Omron Sysmac Studio project python_plc (Sysmac Studio 1.30.0.17, StandardProject)

# Controller new_Controller_0: NX1P2-1140DT1 version 1.13
Axis Sag_kol, settings changed from default: 
Axis Sol_kol, settings changed from default: AxisNumber=1, AxisType=ServoType, UnitsConversion=EnumElement5, UnitsNumerator=8388608, UnitsDenominator=360, MaxVelocity=18000, MaxJogVelocity=18000, MaxPositiveTorqueLimit=350.0, MaxNegativeTorqueLimit=350.0, CountMode=EnumElement2, ModuloMAXPosition=361, ModuloMINPosition=-1, EncoderTypes=Abs
Task PrimaryTask (priority 4, period or condition 2000): Program2
Library MTCP_NJ 1.3. (contents left out)

TYPE Modbus_Data : UNION
    Datas : ARRAY[0..1023] OF word;
    Datas_Dword : ARRAY[0..511] OF DWORD;  (* 4byte *)
    Datas_Lword : ARRAY[0..255] OF lword;  (* 8 byte *)
END_UNION END_TYPE
TYPE Servo : STRUCT
    mc_pwr_ready : BOOL;
    mc_pwr_busy : BOOL;
    mc_pwr_err : BOOL;
    mc_pwr_id : WORD;
    jog_positive_enable : BOOL;
    jog_negative_enable : BOOL;
    velocity : LREAL;
    acc_val : LREAL;
    dec_val : LREAL;
    jog_busy : BOOL;
    jog_aborted : BOOL;
    jog_error : BOOL;
    jog_error_id : WORD;
    position_enable : BOOL;
    position_val : LREAL;
    position_direction : _eMC_DIRECTION;
    position_done : BOOL;
    position_busy : BOOL;
    position_active : BOOL;
    position_aborted : BOOL;
    position_err : BOOL;
    position_err_id : word;
    reset_execute : BOOL;
    reset_busy : BOOL;
    reset_failure : BOOL;
    reset_err : BOOL;
    reset_err_id : WORD;
END_STRUCT END_TYPE
TYPE Srv : STRUCT
    Axis : _sAXIS_REF;
    pwr_enable : BOOL;
    pwr_busy : BOOL;
    pwr_err : BOOL;
    pwr_errid : WORD;
    pwr_status : BOOL;
    rst_enable : BOOL;
    rst_busy : BOOL;
    rst_failure : BOOL;
    rst_err : BOOL;
    rst_errid : WORD;
    rst_done : BOOL;
    parameter : _sAXIS_PARAM;
    read_enable : BOOL;
    read_busy : BOOL;
    read_aborted : BOOL;
    read_err : BOOL;
    read_errid : WORD;
    read_done : BOOL;
    move_enable : BOOL;
    move_position : LREAL;
    move_velocity : LREAL;
    move_acc : LREAL;
    move_dcc : LREAL;
    move_jerk : LREAL;
    move_direction : _eMC_DIRECTION;
    move_buffermode : _eMC_BUFFER_MODE;
    move_mode : _eMC_MOVE_MODE;
    move_busy : BOOL;
    move_active : BOOL;
    move_aborted : BOOL;
    move_err : BOOL;
    move_errid : WORD;
    move_done : BOOL;
    jog_pos_enable : BOOL;
    jog_neg_enable : BOOL;
    jog_velocity : LREAL;
    jog_acc : LREAL;
    jog_dcc : LREAL;
    jog_busy : bool;
    jog_aborted : bool;
    jog_err : bool;
    jog_errid : WORD;
    jog_errid_Copy : WORD;
    move_velocity_enable : BOOL;
    move_velocity_position : LREAL;
    move_velocity_velocity : LREAL;
    move_velocity_acc : LREAL;
    move_velocity_dcc : LREAL;
    move_velocity_jerk : LREAL;
    move_velocity_direction : _eMC_DIRECTION;
    move_velocity_buffermode : _eMC_BUFFER_MODE;
    move_velocity_continous : bool;
    move_velocity_busy : BOOL;
    move_velocity_active : BOOL;
    move_velocity_aborted : BOOL;
    move_velocity_err : BOOL;
    move_velocity_errid : WORD;
    move_velocity_done : BOOL;
    servo_start : BOOL;
    sync_move_start : bool;
    sync_move_buffer : _eMC_BUFFER_MODE;
    sync_move_inPosition : bool;
    sync_move_busy : bool;
    sync_move_active : bool;
    sync_move_aborted : bool;
    sync_move_error : bool;
    sync_move_errorid : WORD;
    sync_move_relative_start : bool;
    sync_move_relative_buffer : _eMC_BUFFER_MODE;
    sync_move_relative_invelocity : bool;
    sync_move_relative_active : bool;
    sync_move_relative_busy : bool;
    sync_move_relative_aborted : bool;
    sync_move_relative_error : bool;
    sync_move_relative_errorid : WORD;
    sync_move_relative_mode : _eMC_CMDPOS_MODE;
END_STRUCT END_TYPE
TYPE UDP_Data : UNION
    bytes : ARRAY[0..1999] OF BYTE;
    words : ARRAY[0..999] OF WORD;
    dwords : ARRAY[0..499] OF DWORD;
    lwords : ARRAY[0..249] OF LWORD;
END_UNION END_TYPE

VAR_GLOBAL CONSTANT
    Sol_kol : _sAXIS_REF;  (* at MC://_MC_AX[1] *)
END_VAR
VAR_GLOBAL
    register_array : Modbus_Data;
    Sistem_start : BOOL;  (* at BuiltInIO://cpu/#0/Input_Bit_00 *)
    Sistem_stop : BOOL;  (* at BuiltInIO://cpu/#0/Input_Bit_01 *)
    Reset : BOOL;  (* at BuiltInIO://cpu/#0/Input_Bit_02 *)
    Acil_Stop : BOOL;  (* at BuiltInIO://cpu/#0/Input_Bit_03 *)
END_VAR
VAR_GLOBAL CONSTANT
    Sag_kol : _sAXIS_REF;  (* at MC://_MC_AX[0] *)
END_VAR
VAR_GLOBAL
    statusword_s1 : WORD;  (* at ECAT://node#1/Statusword *)
    error_code_s1 : WORD;  (* at ECAT://node#1/Error code *)
    pos_act_s1 : DINT;  (* at ECAT://node#1/Position actual value *)
    trq_act_s1 : INT;  (* at ECAT://node#1/Torque actual value *)
    mode_s1 : SINT;  (* at ECAT://node#1/Modes of operation display *)
    digital_inputs_s1 : DWORD;  (* at ECAT://node#1/Digital inputs *)
END_VAR

PROGRAM Program0
VAR
    start : BOOL;
    sistem_calisiyor : BOOL;
    stop : BOOL;
    reset : BOOL;
    tcp_port_no : UINT := 0;
    tcp_port_add : STRING[15] := '192.168.0.100';
    dst_port : UINT := 6000;
    Trigger : BOOL;
    MTCP_Server_fc : MTCP_Server;
    Register_Modbus : ARRAY[0..1023] OF LREAL;
    coils : ARRAY[0..1023] OF BOOL;
    baglan2 : BOOL;
    MTCP_Client_Fn06_fb : MTCP_Client_Fn06;
    say : INT;
    ARADEGER : WORD;
    ARA2 : INT;
    fccnt : CTU;
    Servo_1_Hazir : BOOL;
    Servo_2_Hazir : bool;
    servo1_pwr : MC_Power;
    servo1_jog_fc : MC_MoveJog;
    servo1_move_abs_fc : MC_MoveAbsolute;
    servo2_pwr : MC_Power;
    servo2_move_abs_fc : MC_MoveAbsolute;
    servo1_reset_fc : MC_Reset;
    servo2_reset_fc : MC_Reset;
    baglan : bool;
    Register_Modbus_real : ARRAY[0..1023] OF real;
    ara : LINT;
    servo2_jog_fc : MC_MoveJog;
    run : BOOL;
    i : INT;
    tmp : LREAL;
    whatcdog : WORD := 9999;
    TCP_error : BOOL;
    TCP_ID : WORD;
    TCP_status : _eCONNECTION_STATE;
    tmp2 : LWORD;
    Status_notconnected : _eCONNECTION_STATE := _ESTABLISHED;
    fc_ton : TON;
    fc_ton1 : TON;
    fc_set : RS;
    fc_sr : SR;
    c : BOOL;
    testttt : REAL;
    testtlreal : LREAL;
    sol_eksen : Servo;
    sag_eksen : Servo;
    serv1_not_busy : BOOL;
    i_syc : INT;
    tmp3 : REAL;
    sol_kol_parameter : _sAXIS_PARAM;
    mc_readPara_sol : MC_ReadAxisParameter;
    sol_eksen_mcread_busy : BOOL;
    sol_eksen_mcread_aborted : BOOL;
    sol_eksen_mcread_error : BOOL;
    sol_eksen_mcread_errid : WORD;
END_VAR
VAR_EXTERNAL CONSTANT
    Sol_kol : _sAXIS_REF;
END_VAR
VAR_EXTERNAL
    register_array : Modbus_Data;
    Sistem_start : BOOL;
    Acil_Stop : BOOL;
    Sistem_stop : BOOL;
END_VAR
VAR_EXTERNAL CONSTANT
    Sag_kol : _sAXIS_REF;
END_VAR
VAR
    _p1 : BOOL;
    _p2 : BOOL;
    _p3 : BOOL;
    _p4 : BOOL;
    _p5 : BOOL;
    _e6 : R_TRIG;
END_VAR

(* Section Servo_Kontrol: ladder, written here as Structured Text *)

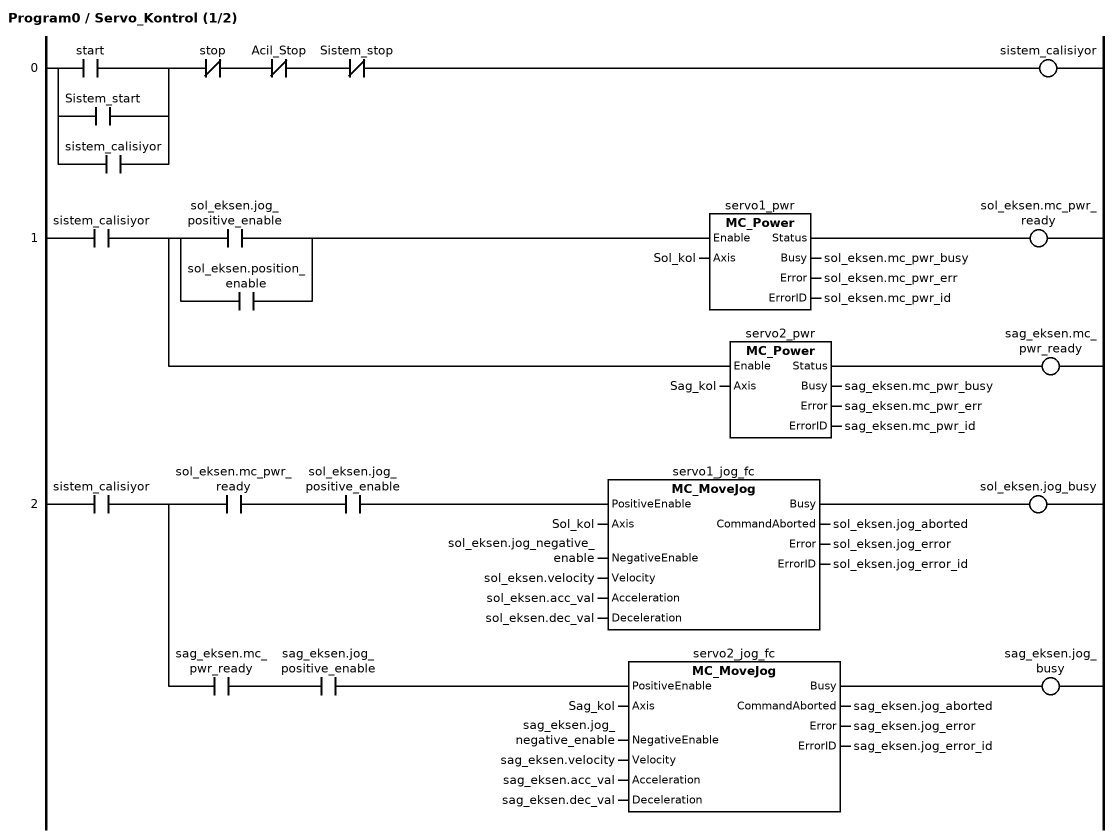
(* Rung 0 *)
sistem_calisiyor := (start OR Sistem_start OR sistem_calisiyor) AND NOT stop AND NOT Acil_Stop AND NOT Sistem_stop;
(* Rung 1 *)
_p1 := sistem_calisiyor AND (sol_eksen.jog_positive_enable OR sol_eksen.position_enable);
servo1_pwr(Enable := _p1, Axis := Sol_kol, Busy => sol_eksen.mc_pwr_busy, Error => sol_eksen.mc_pwr_err, ErrorID => sol_eksen.mc_pwr_id);
sol_eksen.mc_pwr_ready := servo1_pwr.Status;
servo2_pwr(Enable := sistem_calisiyor, Axis := Sag_kol, Busy => sag_eksen.mc_pwr_busy, Error => sag_eksen.mc_pwr_err, ErrorID => sag_eksen.mc_pwr_id);
sag_eksen.mc_pwr_ready := servo2_pwr.Status;
(* Rung 2 *)
_p2 := sistem_calisiyor AND sol_eksen.mc_pwr_ready AND sol_eksen.jog_positive_enable;
servo1_jog_fc(PositiveEnable := _p2, Axis := Sol_kol, NegativeEnable := sol_eksen.jog_negative_enable, Velocity := sol_eksen.velocity, Acceleration := sol_eksen.acc_val, Deceleration := sol_eksen.dec_val, CommandAborted => sol_eksen.jog_aborted, Error => sol_eksen.jog_error, ErrorID => sol_eksen.jog_error_id);
sol_eksen.jog_busy := servo1_jog_fc.Busy;
_p3 := sistem_calisiyor AND sag_eksen.mc_pwr_ready AND sag_eksen.jog_positive_enable;
servo2_jog_fc(PositiveEnable := _p3, Axis := Sag_kol, NegativeEnable := sag_eksen.jog_negative_enable, Velocity := sag_eksen.velocity, Acceleration := sag_eksen.acc_val, Deceleration := sag_eksen.dec_val, CommandAborted => sag_eksen.jog_aborted, Error => sag_eksen.jog_error, ErrorID => sag_eksen.jog_error_id);
sag_eksen.jog_busy := servo2_jog_fc.Busy;

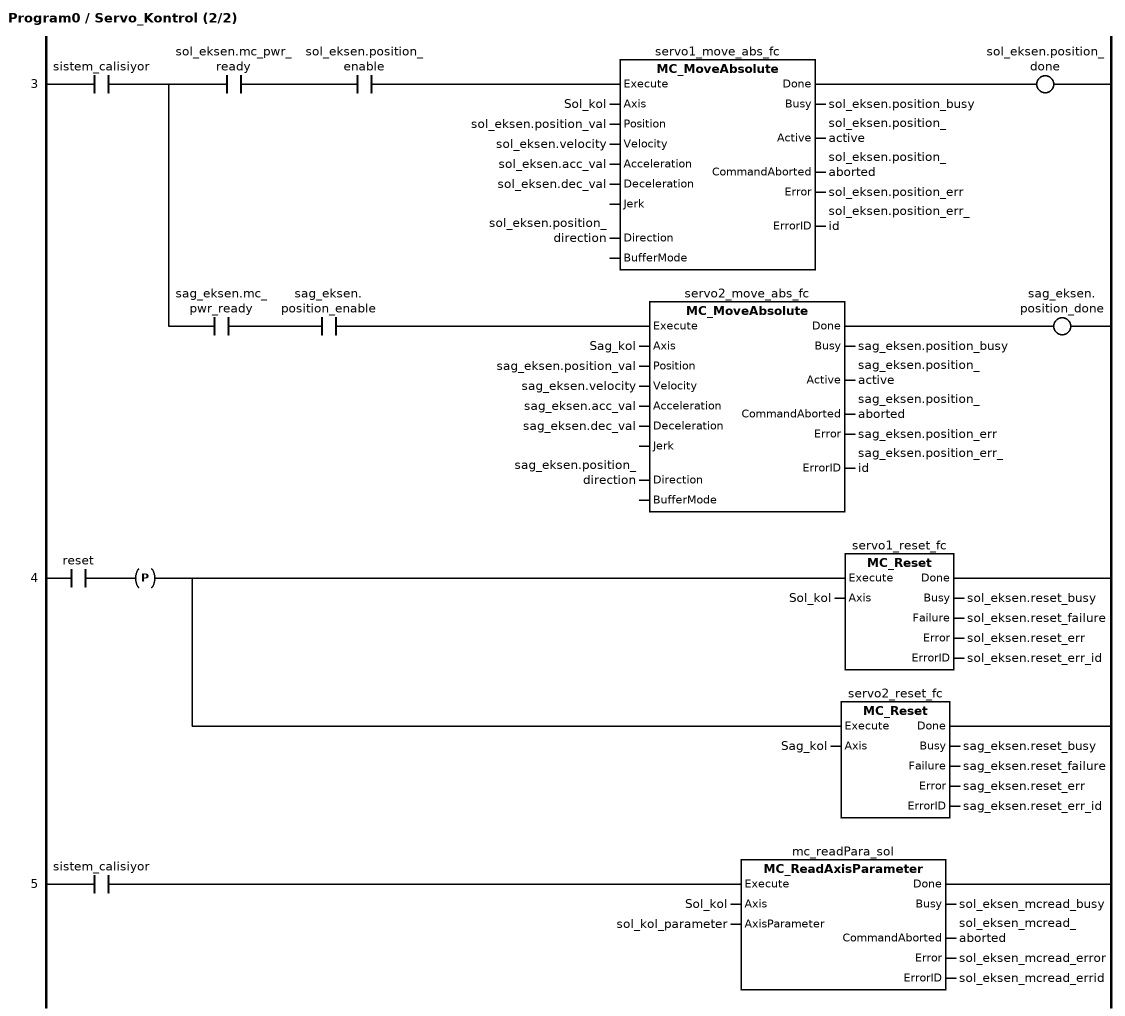
(* Rung 3 *)
_p4 := sistem_calisiyor AND sol_eksen.mc_pwr_ready AND sol_eksen.position_enable;
servo1_move_abs_fc(Execute := _p4, Axis := Sol_kol, Position := sol_eksen.position_val, Velocity := sol_eksen.velocity, Acceleration := sol_eksen.acc_val, Deceleration := sol_eksen.dec_val, Direction := sol_eksen.position_direction, Busy => sol_eksen.position_busy, Active => sol_eksen.position_active, CommandAborted => sol_eksen.position_aborted, Error => sol_eksen.position_err, ErrorID => sol_eksen.position_err_id);
sol_eksen.position_done := servo1_move_abs_fc.Done;
_p5 := sistem_calisiyor AND sag_eksen.mc_pwr_ready AND sag_eksen.position_enable;
servo2_move_abs_fc(Execute := _p5, Axis := Sag_kol, Position := sag_eksen.position_val, Velocity := sag_eksen.velocity, Acceleration := sag_eksen.acc_val, Deceleration := sag_eksen.dec_val, Direction := sag_eksen.position_direction, Busy => sag_eksen.position_busy, Active => sag_eksen.position_active, CommandAborted => sag_eksen.position_aborted, Error => sag_eksen.position_err, ErrorID => sag_eksen.position_err_id);
sag_eksen.position_done := servo2_move_abs_fc.Done;
(* Rung 4 *)
_e6(CLK := reset);
servo1_reset_fc(Execute := _e6.Q, Axis := Sol_kol, Busy => sol_eksen.reset_busy, Failure => sol_eksen.reset_failure, Error => sol_eksen.reset_err, ErrorID => sol_eksen.reset_err_id);
servo2_reset_fc(Execute := _e6.Q, Axis := Sag_kol, Busy => sag_eksen.reset_busy, Failure => sag_eksen.reset_failure, Error => sag_eksen.reset_err, ErrorID => sag_eksen.reset_err_id);
(* Rung 5 *)
mc_readPara_sol(Execute := sistem_calisiyor, Axis := Sol_kol, AxisParameter := sol_kol_parameter, Busy => sol_eksen_mcread_busy, CommandAborted => sol_eksen_mcread_aborted, Error => sol_eksen_mcread_error, ErrorID => sol_eksen_mcread_errid);

(* Section tcp_COM: ladder, written here as Structured Text *)

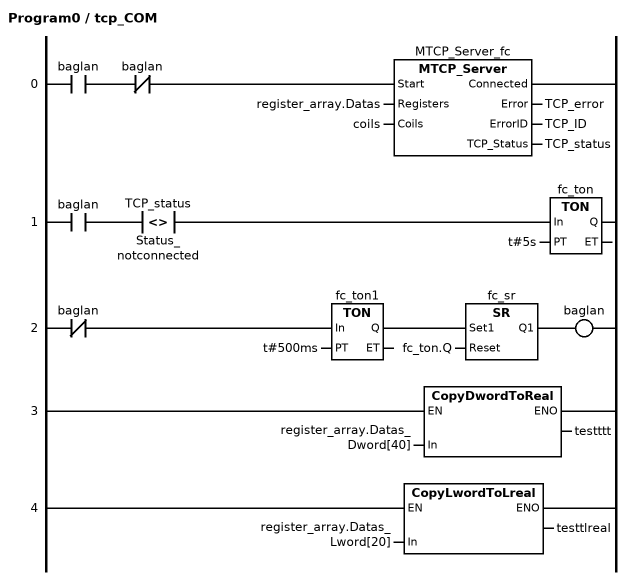
(* Rung 0 *)
MTCP_Server_fc(Start := baglan AND NOT baglan, Registers := register_array.Datas, Coils := coils, Error => TCP_error, ErrorID => TCP_ID, TCP_Status => TCP_status);
(* Rung 1 *)
fc_ton(In := baglan AND (TCP_status <> Status_notconnected), PT := t#5s);
(* Rung 2 *)
fc_ton1(In := NOT baglan, PT := t#500ms);
fc_sr(Set1 := fc_ton1.Q, Reset := fc_ton.Q);
baglan := fc_sr.Q1;
(* Rung 3 *)
testttt := CopyDwordToReal(In := register_array.Datas_Dword[40]);
(* Rung 4 *)
testtlreal := CopyLwordToLreal(In := register_array.Datas_Lword[20]);

(* Section Data_move: ladder, written here as Structured Text *)

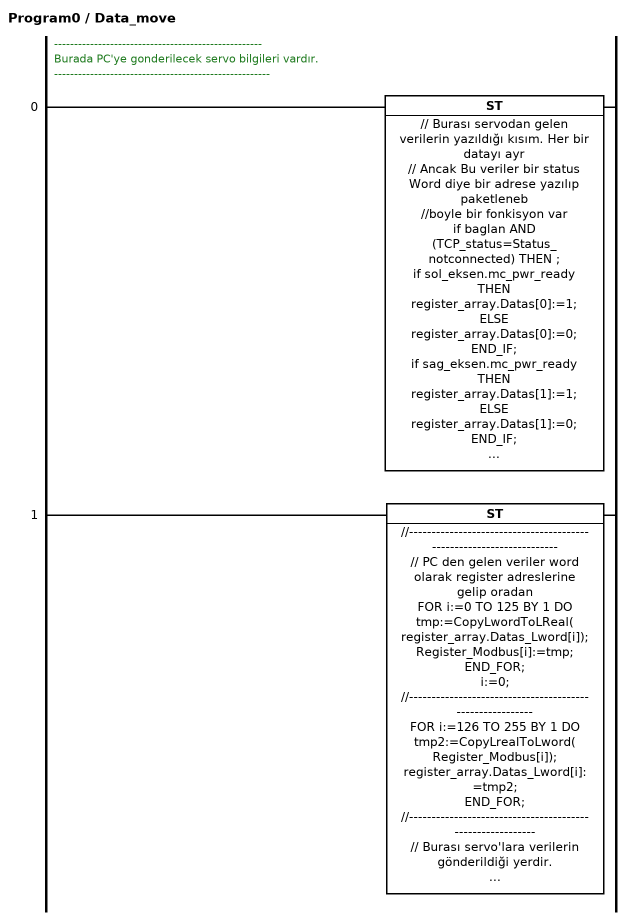
(* Rung 0: ---------------------------------------------------- / Burada PC'ye gonderilecek servo bilgileri vardır. / ------------------------------------------------------ *)
// Burası servodan gelen verilerin yazıldığı kısım. Her bir datayı ayro word'lere gonderildi 
// Ancak Bu veriler bir status Word diye bir adrese yazılıp paketlenebilir. Bunun için bit olarak o wordun ilgili adresine bit yazmak gerekiyor 
//boyle bir fonkisyon var

if baglan AND (TCP_status=Status_notconnected) THEN ;
	if sol_eksen.mc_pwr_ready THEN 
		register_array.Datas[0]:=1; 
	ELSE
		register_array.Datas[0]:=0;
	END_IF;
		if sag_eksen.mc_pwr_ready THEN 
		register_array.Datas[1]:=1; 
	ELSE
		register_array.Datas[1]:=0;
	END_IF;
	if sol_eksen.position_done THEN 
		register_array.Datas[2]:=1; 
	ELSE
		register_array.Datas[2]:=0;
	END_IF;
	if sag_eksen.position_done THEN 
		register_array.Datas[3]:=1; 
	ELSE
		register_array.Datas[3]:=0;
	END_IF;
	if sol_eksen.jog_busy OR sol_eksen.mc_pwr_busy OR sol_eksen.position_busy OR sol_eksen.reset_busy THEN 
		register_array.Datas[4]:=1; 
	ELSE
		register_array.Datas[4]:=0;
	END_IF;
	if sag_eksen.jog_busy OR sag_eksen.mc_pwr_busy OR sag_eksen.position_busy OR sag_eksen.reset_busy THEN 
		register_array.Datas[5]:=1; 
	ELSE
		register_array.Datas[5]:=0;
	END_IF;
	
	// Eger herhangi bir bloktan hata geliyor ise burada o bloktan gelen hata mesajı goruntulenir
	//-----------Servo-1------------------------------------------------------------------------------//
	if sol_eksen.jog_error THEN 
		register_array.Datas[6]:=sol_eksen.jog_error_id;
	ELSIF sol_eksen.mc_pwr_err THEN
		register_array.Datas[6]:=sol_eksen.mc_pwr_id;
	ELSIF sol_eksen.position_err THEN 
		register_array.Datas[6]:=sol_eksen.position_err_id;
	ELSIF sol_eksen.reset_err THEN
		register_array.Datas[6]:=sol_eksen.reset_err_id;
	END_IF;
	//-----------Servo-2------------------------------------------------------------------------------//
	if sag_eksen.jog_error THEN 
		register_array.Datas[7]:=sag_eksen.jog_error_id;
	ELSIF sag_eksen.mc_pwr_err THEN
		register_array.Datas[7]:=sag_eksen.mc_pwr_id;
	ELSIF sag_eksen.position_err THEN 
		register_array.Datas[7]:=sag_eksen.position_err_id;
	ELSIF sag_eksen.reset_err THEN
		register_array.Datas[7]:=sag_eksen.reset_err_id;
	END_IF;

// Eger baglantı yok ise tum gonderilen degerleri sıfırlar suan icin 10 word adresi sıfırladım
	//---------------------------------------------------------------------------------------------//
ELSE;
		
	FOR i_syc:=0 TO 10 BY 1 DO
		
		register_array.Datas[i]:=0;
	END_FOR;
	
END_IF;
		
		
(* Rung 1 *)
//---------------------------------------------------------------------------------------------------------
// PC den gelen veriler word olarak register adreslerine gelip oradan LREAL olarak kaydediliyor
FOR i:=0 TO 125 BY 1 DO

tmp:=CopyLwordToLReal(register_array.Datas_Lword[i]);

Register_Modbus[i]:=tmp;

END_FOR; 
i:=0;

//---------------------------------------------------------
FOR i:=126 TO 255 BY 1 DO

tmp2:=CopyLrealToLword(Register_Modbus[i]);
register_array.Datas_Lword[i]:=tmp2;

END_FOR; 
//----------------------------------------------------------
// Burası servo'lara verilerin gönderildiği yerdir.
// Register modbus alanı Lreal olarak tanımlıdır. 
// bu adresler 8 byte tır adreslemesi de buna göre yapılmıstır
if sistem_calisiyor and baglan THEN 
	sol_eksen.acc_val:=Register_Modbus[20];
	sag_eksen.acc_val:=Register_Modbus[21];
	sol_eksen.dec_val:=Register_Modbus[22];
	sag_eksen.dec_val:=Register_Modbus[23];
	sol_eksen.position_val:=Register_Modbus[24];
	sag_eksen.position_val:=Register_Modbus[25];
	sol_eksen.velocity:=Register_Modbus[26];
	sag_eksen.velocity:=Register_Modbus[27];
	
	//sol_eksen.position_direction:=register_array.Datas[30]; // Bu iki adreslerin özellikle kontrol edilmesi gerekiyor.
	//sag_eksen.position_direction:=register_array.Datas[31];
	
	
	if register_array.Datas[32]=1 then
	sol_eksen.jog_negative_enable:=1;
	ELSE;
	sol_eksen.jog_negative_enable:=0;
	END_IF;
	
	if register_array.Datas[33]=1 then
	sag_eksen.jog_negative_enable:=1;
	ELSE;
	sag_eksen.jog_negative_enable:=0;
	END_IF;
	
	if register_array.Datas[34]=1 then
	sol_eksen.jog_positive_enable:=1;
	ELSE;
	sol_eksen.jog_positive_enable:=0;
	END_IF;
	
	if register_array.Datas[35]=1 then
	sag_eksen.jog_positive_enable:=1;
	ELSE;
	sag_eksen.jog_positive_enable:=0;
	END_IF;
	
	if register_array.Datas[36]=1 then
	sol_eksen.position_enable:=1;
	ELSE;
	sol_eksen.position_enable:=0;
	END_IF;
	
	if register_array.Datas[37]=1 then
	sag_eksen.position_enable:=1;
	ELSE;
	sag_eksen.position_enable:=0;
	END_IF;
	
	if register_array.Datas[38]=1 then
	Sistem_start:=1;
	ELSE;
	Sistem_start:=0;
	END_IF;

	if register_array.Datas[39]=1 then
	Sistem_stop:=1;
	ELSE;
	Sistem_stop:=0;
	END_IF;
	
	if Register_Modbus[30]=0 THEN
		sol_eksen.jog_positive_enable:=1;
		sag_eksen.jog_positive_enable:=1;
	ELSIF Register_Modbus[30]=1 THEN
	sol_eksen.position_enable:=1;
	sag_eksen.position_enable:=1;
	ELSE;
		sol_eksen.jog_positive_enable:=0;
		sag_eksen.jog_positive_enable:=0;
		sol_eksen.position_enable:=0;
	    sag_eksen.position_enable:=0;
	END_IF;
		
END_IF;
END_PROGRAM

PROGRAM Program1
VAR
    Start : BOOL;
    Stop : BOOL;
    Sistem_Calisiyor : BOOL;
    S1_MC_PWR : MC_Power;
    S1_MC_RESET : MC_Reset;
    S1_MC_ReadAxisParameter : MC_ReadAxisParameter;
    S1_MC_Move : MC_Move;
    S1_MC_MoveJog : MC_MoveJog;
    S1_MC_MoveVelocity : MC_MoveVelocity;
    S1 : Srv;
    coils : ARRAY[0..1023] OF BOOL;
    TCP_error : BOOL;
    TCP_ID : WORD;
    TCP_status : _eCONNECTION_STATE;
    MTCP_Server_fc : MTCP_Server;
    Status_notconnected : _eCONNECTION_STATE := _ESTABLISHED;
    fc_ton : TON;
    fc_ton1 : TON;
    fc_sr : SR;
    TCP_Baglan : BOOL;
    TCP_Register : Modbus_Data;
    tmp_lreal : ARRAY[0..10] OF lreal;
    Register_Modbus : ARRAY[0..1023] OF LREAL;
    tmp_lword : ARRAY[0..10] OF LWORD;
    i : INT;
    testttt : BOOL;
    tmp : ARRAY[0..10] OF INT;
    deneme : ARRAY[0..1023] OF WORD;
END_VAR
VAR_EXTERNAL
    register_array : Modbus_Data;
END_VAR
VAR_EXTERNAL CONSTANT
    Sol_kol : _sAXIS_REF;
END_VAR
VAR
    _p1 : BOOL;
    _p2 : BOOL;
    _p3 : BOOL;
    _p4 : BOOL;
    _p5 : BOOL;
    _p6 : BOOL;
END_VAR

(* Section ServoKontrol2: ladder, written here as Structured Text *)

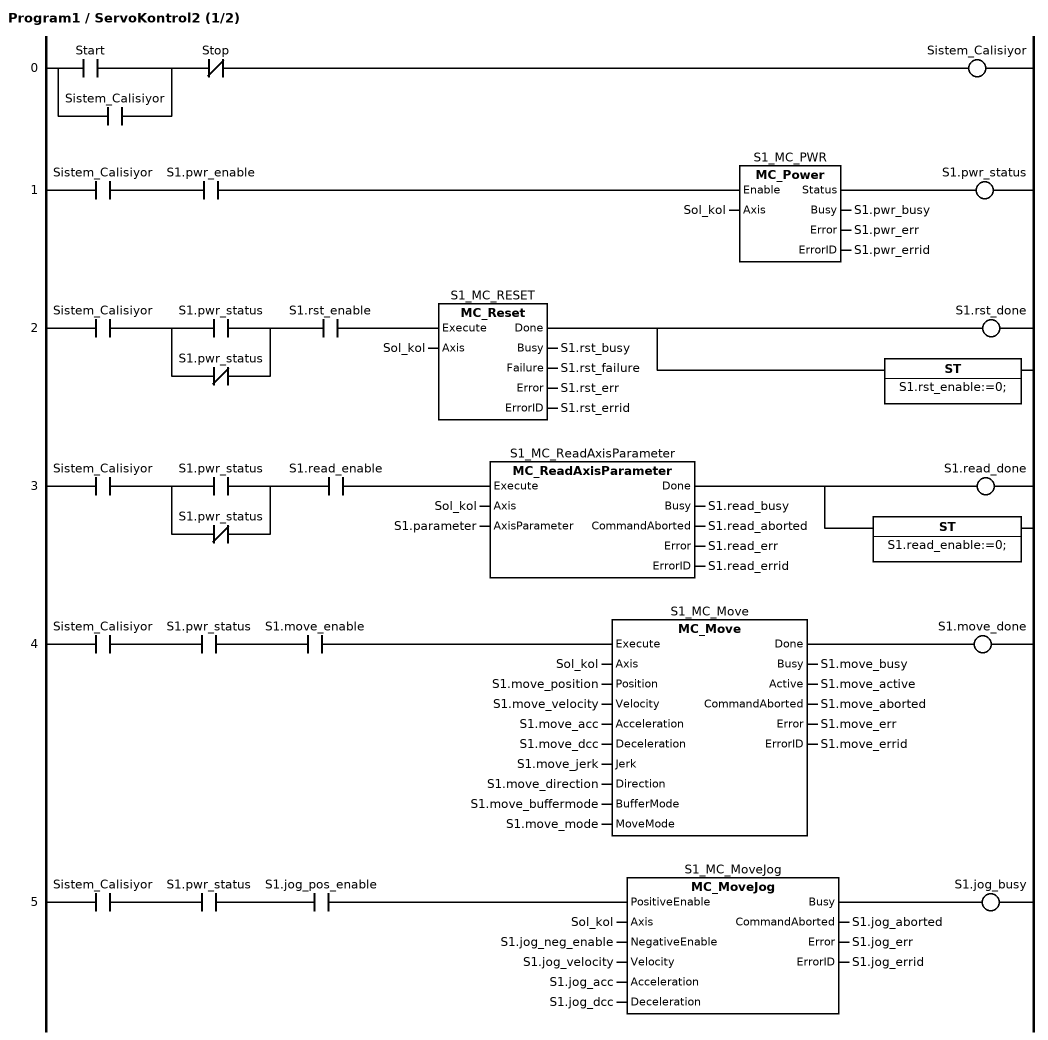
(* Rung 0 *)
Sistem_Calisiyor := (Start OR Sistem_Calisiyor) AND NOT Stop;
(* Rung 1 *)
_p1 := Sistem_Calisiyor AND S1.pwr_enable;
S1_MC_PWR(Enable := _p1, Axis := Sol_kol, Busy => S1.pwr_busy, Error => S1.pwr_err, ErrorID => S1.pwr_errid);
S1.pwr_status := S1_MC_PWR.Status;
(* Rung 2 *)
_p2 := Sistem_Calisiyor AND (S1.pwr_status OR NOT S1.pwr_status) AND S1.rst_enable;
S1_MC_RESET(Execute := _p2, Axis := Sol_kol, Busy => S1.rst_busy, Failure => S1.rst_failure, Error => S1.rst_err, ErrorID => S1.rst_errid);
S1.rst_done := S1_MC_RESET.Done;
IF S1_MC_RESET.Done THEN
    S1.rst_enable:=0;
END_IF;
(* Rung 3 *)
_p3 := Sistem_Calisiyor AND (S1.pwr_status OR NOT S1.pwr_status) AND S1.read_enable;
S1_MC_ReadAxisParameter(Execute := _p3, Axis := Sol_kol, AxisParameter := S1.parameter, Busy => S1.read_busy, CommandAborted => S1.read_aborted, Error => S1.read_err, ErrorID => S1.read_errid);
S1.read_done := S1_MC_ReadAxisParameter.Done;
IF S1_MC_ReadAxisParameter.Done THEN
    S1.read_enable:=0;
END_IF;
(* Rung 4 *)
_p4 := Sistem_Calisiyor AND S1.pwr_status AND S1.move_enable;
S1_MC_Move(Execute := _p4, Axis := Sol_kol, Position := S1.move_position, Velocity := S1.move_velocity, Acceleration := S1.move_acc, Deceleration := S1.move_dcc, Jerk := S1.move_jerk, Direction := S1.move_direction, BufferMode := S1.move_buffermode, MoveMode := S1.move_mode, Busy => S1.move_busy, Active => S1.move_active, CommandAborted => S1.move_aborted, Error => S1.move_err, ErrorID => S1.move_errid);
S1.move_done := S1_MC_Move.Done;
(* Rung 5 *)
_p5 := Sistem_Calisiyor AND S1.pwr_status AND S1.jog_pos_enable;
S1_MC_MoveJog(PositiveEnable := _p5, Axis := Sol_kol, NegativeEnable := S1.jog_neg_enable, Velocity := S1.jog_velocity, Acceleration := S1.jog_acc, Deceleration := S1.jog_dcc, CommandAborted => S1.jog_aborted, Error => S1.jog_err, ErrorID => S1.jog_errid);
S1.jog_busy := S1_MC_MoveJog.Busy;

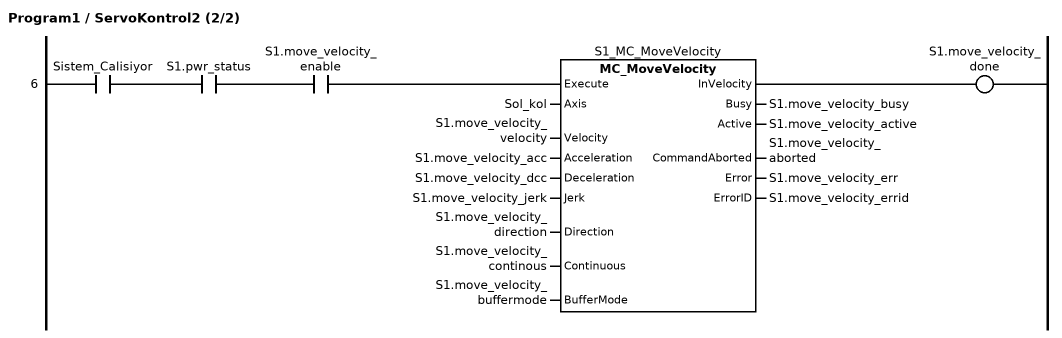
(* Rung 6 *)
_p6 := Sistem_Calisiyor AND S1.pwr_status AND S1.move_velocity_enable;
S1_MC_MoveVelocity(Execute := _p6, Axis := Sol_kol, Velocity := S1.move_velocity_velocity, Acceleration := S1.move_velocity_acc, Deceleration := S1.move_velocity_dcc, Jerk := S1.move_velocity_jerk, Direction := S1.move_velocity_direction, Continuous := S1.move_velocity_continous, BufferMode := S1.move_velocity_buffermode, Busy => S1.move_velocity_busy, Active => S1.move_velocity_active, CommandAborted => S1.move_velocity_aborted, Error => S1.move_velocity_err, ErrorID => S1.move_velocity_errid);
S1.move_velocity_done := S1_MC_MoveVelocity.InVelocity;

(* Section tcp_COM: ladder, written here as Structured Text *)

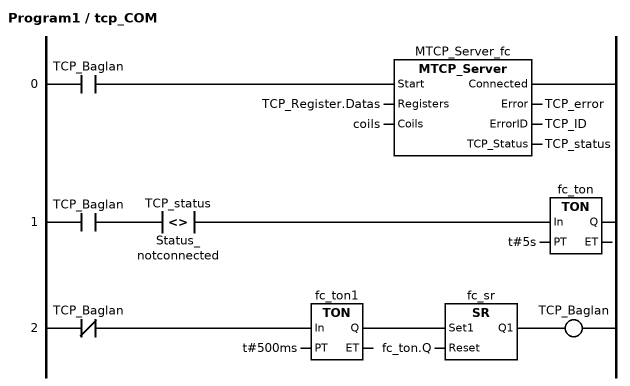
(* Rung 0 *)
MTCP_Server_fc(Start := TCP_Baglan, Registers := TCP_Register.Datas, Coils := coils, Error => TCP_error, ErrorID => TCP_ID, TCP_Status => TCP_status);
(* Rung 1 *)
fc_ton(In := TCP_Baglan AND (TCP_status <> Status_notconnected), PT := t#5s);
(* Rung 2 *)
fc_ton1(In := NOT TCP_Baglan, PT := t#500ms);
fc_sr(Set1 := fc_ton1.Q, Reset := fc_ton.Q);
TCP_Baglan := fc_sr.Q1;

(* Section Data_Move: ladder, written here as Structured Text *)

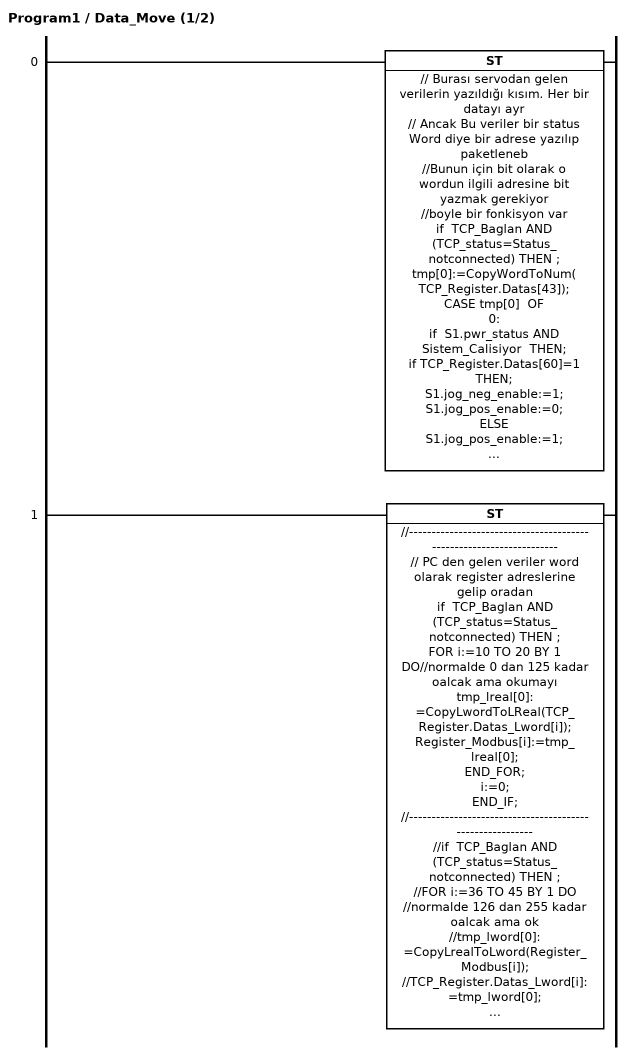
(* Rung 0 *)
// Burası servodan gelen verilerin yazıldığı kısım. Her bir datayı ayro word'lere gonderildi 
// Ancak Bu veriler bir status Word diye bir adrese yazılıp paketlenebilir. 
//Bunun için bit olarak o wordun ilgili adresine bit yazmak gerekiyor 
//boyle bir fonkisyon var

if  TCP_Baglan AND (TCP_status=Status_notconnected) THEN ;

	tmp[0]:=CopyWordToNum(TCP_Register.Datas[43]);
	CASE tmp[0]  OF
    0:
            if  S1.pwr_status AND Sistem_Calisiyor  THEN;
				if TCP_Register.Datas[60]=1  THEN;
					S1.jog_neg_enable:=1;
					S1.jog_pos_enable:=0;
				ELSE
					S1.jog_pos_enable:=1;
					S1.jog_neg_enable:=0;
				END_IF;
			ELSE;
				S1.jog_pos_enable:=0;
				S1.jog_neg_enable:=0;	
			END_IF;	
			
			S1.move_enable:=0;
			S1.move_mode:=_mcAbsolute;
			S1.move_velocity_enable:=0;
    16368:
            S1.move_enable:=1;
			S1.move_mode:=_mcAbsolute;
			S1.jog_pos_enable:=0;
			S1.jog_neg_enable:=0;
			S1.move_velocity_enable:=0;
	16384:
			S1.move_enable:=1;
			S1.move_mode:=_mcRelative;
			S1.jog_pos_enable:=0;
			S1.jog_neg_enable:=0;
			S1.move_velocity_enable:=0;
	16392:
			S1.move_velocity_enable:=1;
       		S1.move_enable:=0;
			S1.move_mode:=_mcAbsolute;
			S1.jog_pos_enable:=0;
			S1.jog_neg_enable:=0;
	ELSE
		    S1.jog_pos_enable:=0;
			S1.jog_neg_enable:=0;
			S1.move_enable:=0;
			S1.move_mode:=_mcAbsolute;
			S1.move_velocity_enable:=0;
    
	END_CASE;
	if TCP_Register.Datas[44]=1 THEN;
			S1.pwr_enable:=1; 
		ELSE
			S1.pwr_enable:=0;
		END_IF;
	S1.move_velocity:=Register_Modbus[12];S1.jog_velocity:=S1.move_velocity;S1.move_velocity_velocity:=S1.move_velocity;
	S1.move_acc:=Register_Modbus[13];S1.jog_acc:=S1.move_acc;S1.move_velocity_acc:=S1.move_acc;
	S1.move_dcc:=Register_Modbus[14];S1.jog_dcc:=S1.move_dcc;S1.move_velocity_dcc:=S1.move_dcc;
	S1.move_position:=Register_Modbus[16];
	if TCP_Register.Datas[40]=1 THEN;
		S1.move_direction:=_mcNegativeDirection;
		S1.move_velocity_direction:=_mcNegativeDirection;
	ELSE
		S1.move_direction:=_mcPositiveDirection;
		S1.move_velocity_direction:=_mcPositiveDirection;
	END_IF;
	if TCP_Register.Datas[72]=1 THEN;
		S1.rst_enable:=1;
	ELSE
		S1.rst_enable:=0;
	END_IF;
END_IF;
(* Rung 1 *)
//---------------------------------------------------------------------------------------------------------
// PC den gelen veriler word olarak register adreslerine gelip oradan LREAL olarak kaydediliyor
if  TCP_Baglan AND (TCP_status=Status_notconnected) THEN ;
	FOR i:=10 TO 20 BY 1 DO//normalde 0 dan 125 kadar oalcak ama okumayı hızlandırmak için azalttım

	tmp_lreal[0]:=CopyLwordToLReal(TCP_Register.Datas_Lword[i]);

	Register_Modbus[i]:=tmp_lreal[0];

	END_FOR; 
	i:=0;
END_IF;

//---------------------------------------------------------
//if  TCP_Baglan AND (TCP_status=Status_notconnected) THEN ;
	//FOR i:=36 TO 45 BY 1 DO //normalde 126 dan 255 kadar oalcak ama okumayı hızlandırmak için azalttım

	//tmp_lword[0]:=CopyLrealToLword(Register_Modbus[i]);
	//TCP_Register.Datas_Lword[i]:=tmp_lword[0];

	//END_FOR;
//END_IF;
//----------------------------------------------------------
// Burası servo'lara verilerin gönderildiği yerdir.
// Register modbus alanı Lreal olarak tanımlıdır. 
// bu adresler 8 byte tır adreslemesi de buna göre yapılmıstır

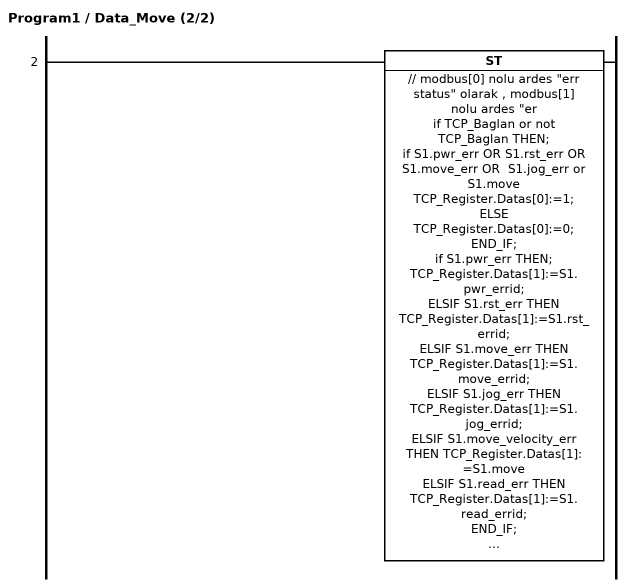
(* Rung 2 *)
// modbus[0] nolu ardes "err status" olarak , modbus[1] nolu ardes "err id" olarak tanımlandı
if TCP_Baglan or not TCP_Baglan THEN;
	if S1.pwr_err OR S1.rst_err OR S1.move_err OR  S1.jog_err or S1.move_velocity_err or S1.read_err THEN;
		TCP_Register.Datas[0]:=1;
	ELSE
		TCP_Register.Datas[0]:=0;
	END_IF;
	if S1.pwr_err THEN; TCP_Register.Datas[1]:=S1.pwr_errid;
	ELSIF S1.rst_err THEN TCP_Register.Datas[1]:=S1.rst_errid;
		ELSIF S1.move_err THEN TCP_Register.Datas[1]:=S1.move_errid;
			ELSIF S1.jog_err THEN TCP_Register.Datas[1]:=S1.jog_errid;
				ELSIF S1.move_velocity_err THEN TCP_Register.Datas[1]:=S1.move_velocity_errid;
					ELSIF S1.read_err THEN TCP_Register.Datas[1]:=S1.read_errid;
	END_IF;
	if s1.pwr_busy OR S1.jog_busy OR S1.move_busy OR S1.move_velocity_busy OR S1.read_busy THEN;
		TCP_Register.Datas[2]:=1;
	ELSE
		TCP_Register.Datas[2]:=0;
	END_IF;
	TCP_Register.Datas[3]:=DINT_TO_WORD( EnumToNum(TCP_status));
	TCP_Register.Datas[4]:=TCP_ID;
		if S1.pwr_status THEN 
		TCP_Register.Datas[5]:=1; 
	ELSE
		TCP_Register.Datas[5]:=0;
	END_IF;
END_IF;
					
		
		
END_PROGRAM

PROGRAM Program2
VAR
    Trigger : bool;  (* Execution condition *)
    DoSendAndRcv : BOOL;  (* Processing *)
    Stage : INT;  (* Stage change *)
    RcvSocketDat : ARRAY[0..1999] OF BYTE := [2000(16#0)];  (* Receive data *)
    WkSocket : _sSOCKET;  (* Socket *)
    SendSocketDat : ARRAY[0..1999] OF BYTE := [2000(16#0)];  (* Send data *)
    SktUDPCreate_instance : SktUDPCreate;
    SktUDPSend_instance : SktUDPSend;
    SktUDPRcv_instance : SktUDPRcv;
    SktClose_instance : SktClose;
    test : SINT;
    test2 : UDP_Data;
    test3 : LREAL;
    test4 : REAL;
    te : DINT;
    test5 : INT;
    test6 : LREAL;
    RcvSocketData : UDP_Data;
    SendSocketData : UDP_Data;
    Start : BOOL;
    Stop : BOOL;
    Sistem_Calisiyor : BOOL;
    S1 : Srv;
    S1_MC_PWR : MC_Power;
    S1_MC_RESET : MC_Reset;
    S1_MC_ReadAxisParameter : MC_ReadAxisParameter;
    S1_MC_Move : MC_Move;
    S1_MC_MoveJog : MC_MoveJog;
    S1_MC_MoveVelocity : MC_MoveVelocity;
    S1_MC_M : MC_SyncMoveAbsolute;
    S1_MC_SyncMoveAbsolute : MC_SyncMoveAbsolute;
    S1_MC_SyncMoveVelocity : MC_SyncMoveVelocity;
    sync_move_relative_start : BOOL;
END_VAR
VAR_EXTERNAL CONSTANT
    _EIP_EtnOnlineSta : BOOL;
END_VAR
VAR_EXTERNAL
    _PowerOnCount : UDINT;
END_VAR
VAR_EXTERNAL CONSTANT
    Sol_kol : _sAXIS_REF;
END_VAR
VAR_EXTERNAL
    error_code_s1 : WORD;
    statusword_s1 : WORD;
    trq_act_s1 : INT;
    mode_s1 : SINT;
    digital_inputs_s1 : DWORD;
    pos_act_s1 : DINT;
END_VAR
VAR
    _p1 : BOOL;
    _p2 : BOOL;
    _p3 : BOOL;
    _p4 : BOOL;
    _p5 : BOOL;
    _p6 : BOOL;
    _p7 : BOOL;
    _p8 : BOOL;
    _p9 : BOOL;
END_VAR

(* Section UDP: ladder, written here as Structured Text *)

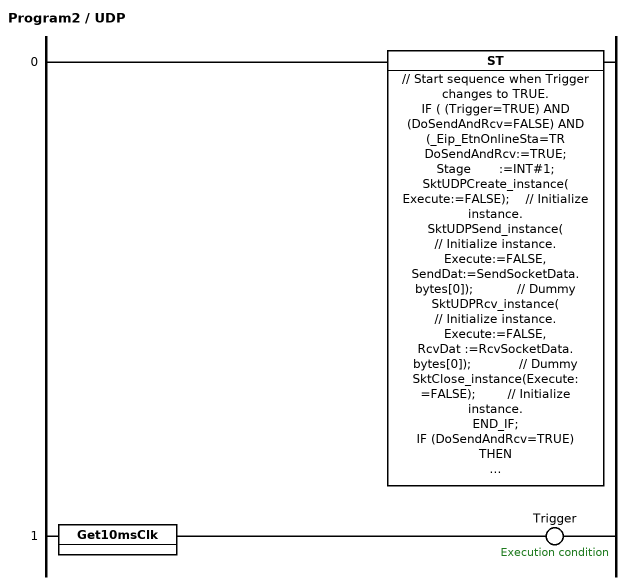
(* Rung 0 *)
// Start sequence when Trigger changes to TRUE.       
IF ( (Trigger=TRUE) AND (DoSendAndRcv=FALSE) AND (_Eip_EtnOnlineSta=TRUE) ) THEN
    DoSendAndRcv:=TRUE;
    Stage       :=INT#1;
    SktUDPCreate_instance(Execute:=FALSE);    // Initialize instance.
    SktUDPSend_instance(                      // Initialize instance.
        Execute:=FALSE,
        SendDat:=SendSocketData.bytes[0]);           // Dummy
    SktUDPRcv_instance(                       // Initialize instance.
        Execute:=FALSE,
        RcvDat :=RcvSocketData.bytes[0]);            // Dummy
    SktClose_instance(Execute:=FALSE);        // Initialize instance.
END_IF;

IF (DoSendAndRcv=TRUE) THEN
    CASE Stage OF
    1 :                                  // Request creating socket.
        SktUDPCreate_instance(
            Execute   :=TRUE,
            SrcUdpPort:=UINT#6000,              // Local UDP port number
            Socket    =>WkSocket);              // Socket

    IF (SktUDPCreate_instance.Done=TRUE) THEN
        Stage:=INT#2;                       // Normal end
    ELSIF (SktUDPCreate_instance.Error=TRUE) THEN
        Stage:=INT#10;                      // Error end
    END_IF;

    2 :                                  // Request sending data
        WkSocket.DstAdr.PortNo:=UINT#6001;
        WkSocket.DstAdr.IpAdr :='192.168.0.100';
        SktUDPSend_instance(
            Execute:=TRUE,
            Socket :=WkSocket,                  // Socket
            SendDat:=SendSocketData.bytes[0],          // Send data
            Size   :=UINT#64);                // Send data size

        IF (SktUDPSend_instance.Done=TRUE) THEN
                Stage:=INT#3;                       // Normal end
        ELSIF (SktUDPSend_instance.Error=TRUE) THEN
                Stage:=INT#20;                      // Error end
        END_IF;

    3 :                                  // Request receiving data.
        SktUDPRcv_instance(
            Execute:=TRUE,
            Socket :=WkSocket,                  // Socket
            TimeOut:=UINT#0,                    // Timeout time
            Size   :=UINT#128,                 // Receive data size
            RcvDat :=RcvSocketData.bytes[0]);          // Receive data

        IF (SktUDPRcv_instance.Done=TRUE) THEN
            Stage:=INT#4;                      // Normal end
        ELSIF (SktUDPRcv_instance.Error=TRUE) THEN
            Stage:=INT#30;                     // Error end
        END_IF;

    4 :                                  // Request closing.
        SktClose_instance(
            Execute:=TRUE,
            Socket :=WkSocket);                 // Socket

        IF (SktClose_instance.Done=TRUE) THEN
            Stage:=INT#0;                       // Normal end
        ELSIF (SktClose_instance.Error=TRUE) THEN
            Stage:=INT#40;                      // Error end
        END_IF;

    0 :                                  // Normal end
        DoSendAndRcv:=FALSE;
        Trigger     :=FALSE;

    ELSE                                 // Interrupted by error.
        DoSendAndRcv:=FALSE;
        Trigger     :=FALSE;
    END_CASE;

END_IF;
(* Rung 1 *)
Trigger := Get10msClk();

(* Section Section0: ladder, written here as Structured Text *)

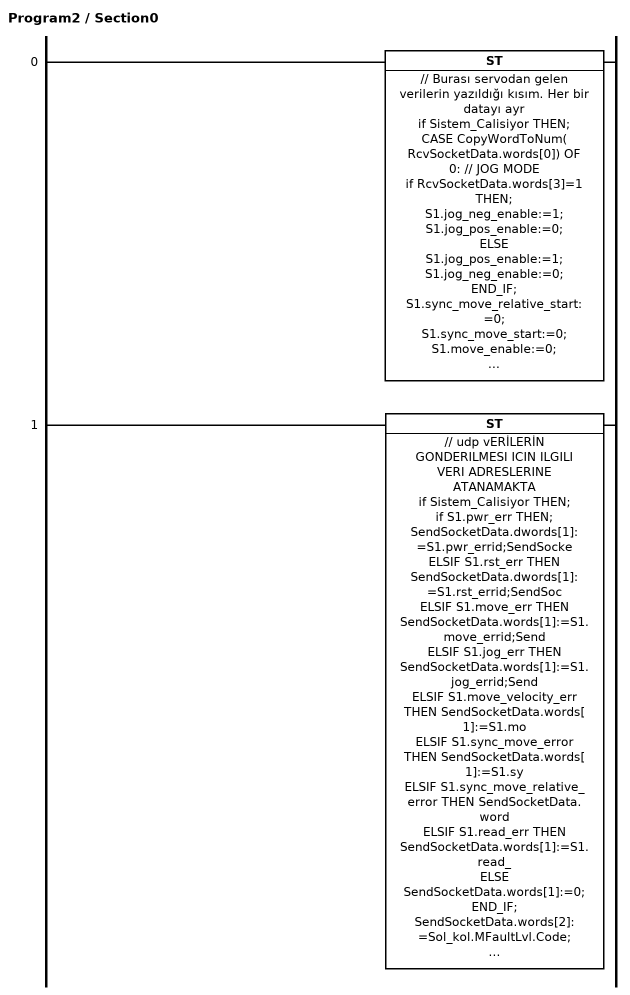
(* Rung 0 *)
// Burası servodan gelen verilerin yazıldığı kısım. Her bir datayı ayro word'lere gonderildi 
if Sistem_Calisiyor THEN;
	CASE CopyWordToNum(RcvSocketData.words[0]) OF
		0: // JOG MODE
		
			if RcvSocketData.words[3]=1  THEN;
				S1.jog_neg_enable:=1;
				S1.jog_pos_enable:=0;
			ELSE
				S1.jog_pos_enable:=1;
				S1.jog_neg_enable:=0;
			END_IF;
		    S1.sync_move_relative_start:=0;
		    S1.sync_move_start:=0;
			S1.move_enable:=0;
			S1.move_mode:=_mcAbsolute;
			S1.move_velocity_enable:=0;
			
		1: // MOVE ABSOLUTE MODE
		S1.move_enable:=1;
			S1.move_mode:=_mcAbsolute;
			S1.jog_pos_enable:=0;
			S1.jog_neg_enable:=0;
			S1.move_velocity_enable:=0;
		2:  // MOVE RELATIVE  MODE
		S1.move_enable:=1;
			S1.move_mode:=_mcRelative;
			S1.jog_pos_enable:=0;
			S1.jog_neg_enable:=0;
			S1.move_velocity_enable:=0;
		3:  // MOVE VELOCITY MODE
		S1.move_velocity_enable:=1;
       		S1.move_enable:=0;
			S1.move_mode:=_mcAbsolute;
			S1.jog_pos_enable:=0;
			S1.jog_neg_enable:=0;
		4:  // MOVE SYNC ABSOLUTE MODE
		S1.sync_move_start:=1;
		S1.sync_move_relative_start:=0;
       		S1.jog_pos_enable:=0;
			S1.jog_neg_enable:=0;
			S1.move_enable:=0;
			S1.move_mode:=_mcAbsolute;
			S1.move_velocity_enable:=0;
			5:  // MOVE SYNC VELOCITY MODE
		S1.sync_move_relative_start:=1;
		S1.sync_move_start:=0;
		S1.jog_pos_enable:=0;
			S1.jog_neg_enable:=0;
			S1.move_enable:=0;
			S1.move_mode:=_mcAbsolute;
			S1.move_velocity_enable:=0;
			S1.jog_pos_enable:=0;
			S1.jog_neg_enable:=0;
	ELSE
		 S1.jog_pos_enable:=0;
		 S1.sync_move_relative_start:=0;
		 S1.sync_move_start:=0;
			S1.jog_neg_enable:=0;
			S1.move_enable:=0;
			S1.move_mode:=_mcAbsolute;
			S1.move_velocity_enable:=0;
	END_CASE;
	if CopyWordToNum(RcvSocketData.words[1])=1 THEN;
			S1.pwr_enable:=1; 
		ELSE
			S1.pwr_enable:=0;
		END_IF;
	S1.move_velocity:=CopyLwordToLreal(RcvSocketData.lwords[2]);
	S1.jog_velocity:=S1.move_velocity;
	S1.move_velocity_velocity:=S1.move_velocity;
	S1.move_velocity_velocity:=S1.move_velocity;
	S1.move_acc:=CopyLwordToLreal(RcvSocketData.lwords[3]);
	S1.jog_acc:=S1.move_acc;S1.move_velocity_acc:=S1.move_acc;
	S1.move_dcc:=CopyLwordToLreal(RcvSocketData.lwords[4]);
	S1.jog_dcc:=S1.move_dcc;S1.move_velocity_dcc:=S1.move_dcc;
	S1.move_position:=CopyLwordToLreal(RcvSocketData.lwords[5]);
	
	if CopyWordToNum(RcvSocketData.words[3])=1 THEN;
		S1.move_direction :=_mcNegativeDirection;
		S1.move_velocity_direction:=_mcNegativeDirection;
	ELSE
		S1.move_direction:=_mcPositiveDirection;
		S1.move_velocity_direction:=_mcPositiveDirection;
	END_IF;
	if CopyWordToNum(RcvSocketData.words[2])=1 THEN;
		S1.rst_enable:=1;
	ELSE
		S1.rst_enable:=0;
	END_IF;
	if CopyWordToNum(RcvSocketData.words[4])=1 THEN;
		S1.servo_start:=1;
	ELSE
		S1.servo_start:=0;
	END_IF;

	
	
END_IF;
(* Rung 1 *)
// udp vERİLERİN GONDERILMESI ICIN ILGILI  VERI ADRESLERINE ATANAMAKTADIR
if Sistem_Calisiyor THEN;
	
	if S1.pwr_err THEN; SendSocketData.dwords[1]:=S1.pwr_errid;SendSocketData.words[0]:=1;
	ELSIF S1.rst_err THEN SendSocketData.dwords[1]:=S1.rst_errid;SendSocketData.words[0]:=2;
		ELSIF S1.move_err THEN SendSocketData.words[1]:=S1.move_errid;SendSocketData.words[0]:=3;
			ELSIF S1.jog_err THEN SendSocketData.words[1]:=S1.jog_errid;SendSocketData.words[0]:=4;
				ELSIF S1.move_velocity_err THEN SendSocketData.words[1]:=S1.move_velocity_errid;SendSocketData.words[0]:=5;
					ELSIF S1.sync_move_error THEN SendSocketData.words[1]:=S1.sync_move_errorid;SendSocketData.words[0]:=6;
						ELSIF S1.sync_move_relative_error THEN SendSocketData.words[1]:=S1.sync_move_relative_errorid;SendSocketData.words[0]:=7;
							ELSIF S1.read_err THEN SendSocketData.words[1]:=S1.read_errid;SendSocketData.words[0]:=8;
	ELSE
		SendSocketData.words[1]:=0;
	END_IF;
	SendSocketData.words[2]:=Sol_kol.MFaultLvl.Code;
	SendSocketData.words[3]:=error_code_s1;
	SendSocketData.words[4]:=statusword_s1;
	SendSocketData.words[5]:=CopyNumToWord(trq_act_s1);
	SendSocketData.words[6]:=CopyNumToWord(mode_s1	);
	if Sol_kol.Dir.Posi THEN;
		SendSocketData.words[7]:=1;
	ELSE
		SendSocketData.words[7]:=0;
	END_IF;
	SendSocketData.dwords[5]:=CopyNumToDword(pos_act_s1);
	SendSocketData.dwords[6]:=digital_inputs_s1;
	
	SendSocketData.lwords[5]:=CopyLrealToLword(Sol_kol.Cmd.Vel);
	SendSocketData.lwords[6]:=CopyLrealToLword(Sol_kol.Cmd.AccDec);
	SendSocketData.lwords[7]:=CopyLrealToLword(Sol_kol.Cmd.Pos);
	SendSocketData.lwords[8]:=CopyLrealToLword(Sol_kol.Cmd.Trq);
	
	
END_IF;

(* Section ServoKontrol2: ladder, written here as Structured Text *)

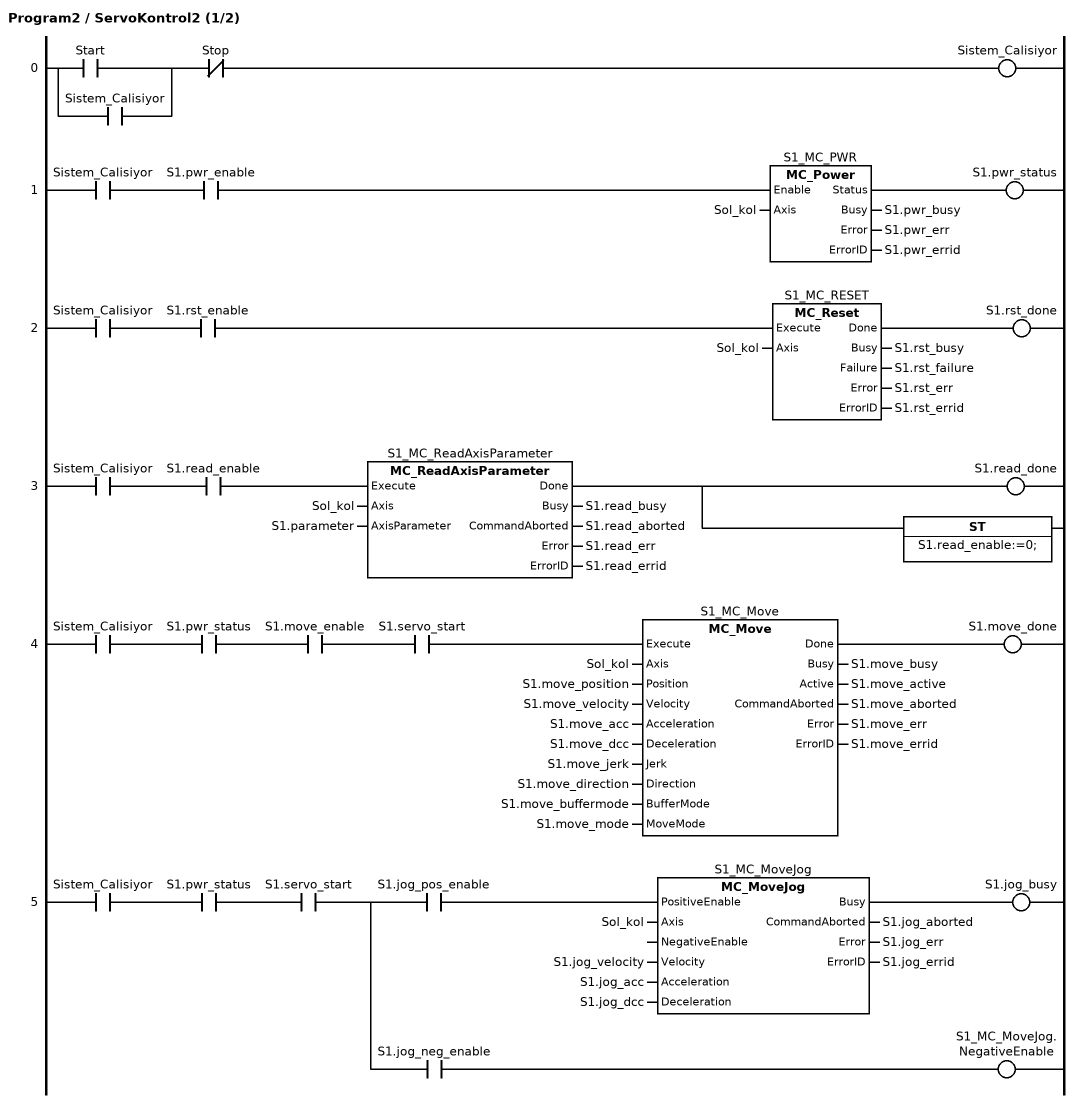
(* Rung 0 *)
Sistem_Calisiyor := (Start OR Sistem_Calisiyor) AND NOT Stop;
(* Rung 1 *)
_p1 := Sistem_Calisiyor AND S1.pwr_enable;
S1_MC_PWR(Enable := _p1, Axis := Sol_kol, Busy => S1.pwr_busy, Error => S1.pwr_err, ErrorID => S1.pwr_errid);
S1.pwr_status := S1_MC_PWR.Status;
(* Rung 2 *)
_p2 := Sistem_Calisiyor AND S1.rst_enable;
S1_MC_RESET(Execute := _p2, Axis := Sol_kol, Busy => S1.rst_busy, Failure => S1.rst_failure, Error => S1.rst_err, ErrorID => S1.rst_errid);
S1.rst_done := S1_MC_RESET.Done;
(* Rung 3 *)
_p3 := Sistem_Calisiyor AND S1.read_enable;
S1_MC_ReadAxisParameter(Execute := _p3, Axis := Sol_kol, AxisParameter := S1.parameter, Busy => S1.read_busy, CommandAborted => S1.read_aborted, Error => S1.read_err, ErrorID => S1.read_errid);
S1.read_done := S1_MC_ReadAxisParameter.Done;
IF S1_MC_ReadAxisParameter.Done THEN
    S1.read_enable:=0;
END_IF;
(* Rung 4 *)
_p4 := Sistem_Calisiyor AND S1.pwr_status AND S1.move_enable AND S1.servo_start;
S1_MC_Move(Execute := _p4, Axis := Sol_kol, Position := S1.move_position, Velocity := S1.move_velocity, Acceleration := S1.move_acc, Deceleration := S1.move_dcc, Jerk := S1.move_jerk, Direction := S1.move_direction, BufferMode := S1.move_buffermode, MoveMode := S1.move_mode, Busy => S1.move_busy, Active => S1.move_active, CommandAborted => S1.move_aborted, Error => S1.move_err, ErrorID => S1.move_errid);
S1.move_done := S1_MC_Move.Done;
(* Rung 5 *)
_p5 := Sistem_Calisiyor AND S1.pwr_status AND S1.servo_start;
_p6 := _p5 AND S1.jog_pos_enable;
S1_MC_MoveJog(PositiveEnable := _p6, Axis := Sol_kol, Velocity := S1.jog_velocity, Acceleration := S1.jog_acc, Deceleration := S1.jog_dcc, CommandAborted => S1.jog_aborted, Error => S1.jog_err, ErrorID => S1.jog_errid);
S1.jog_busy := S1_MC_MoveJog.Busy;
S1_MC_MoveJog.NegativeEnable := _p5 AND S1.jog_neg_enable;

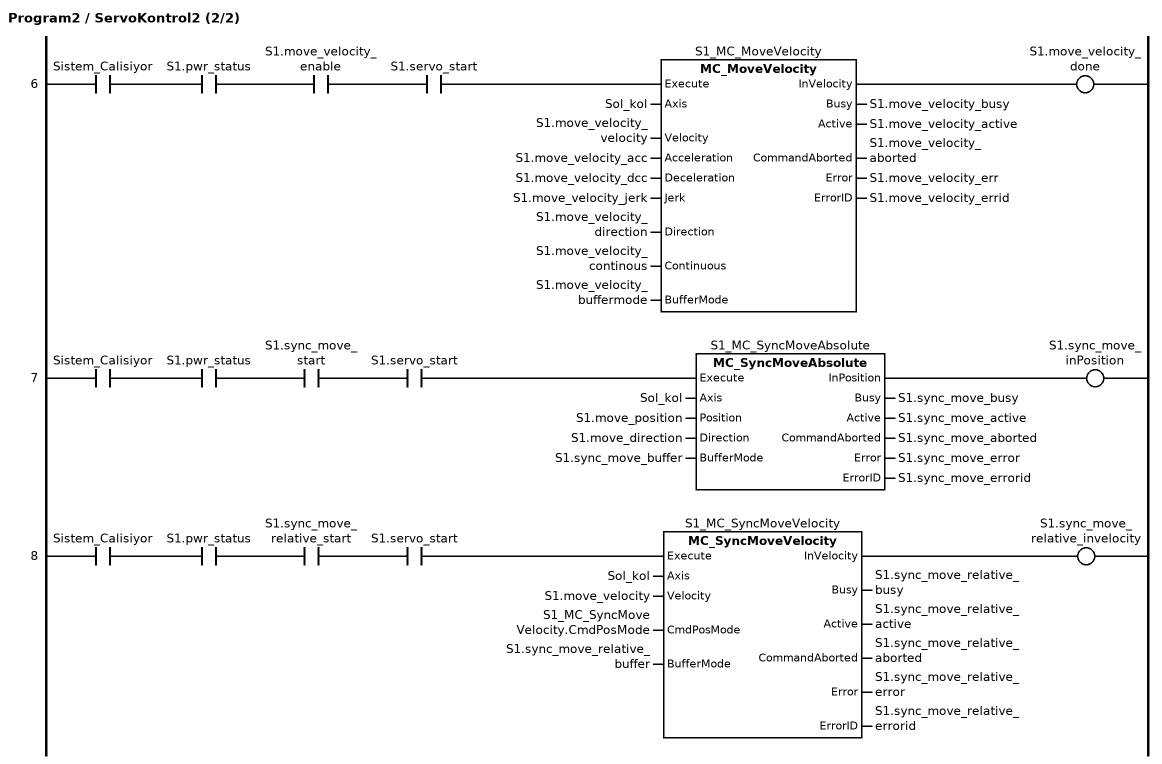
(* Rung 6 *)
_p7 := Sistem_Calisiyor AND S1.pwr_status AND S1.move_velocity_enable AND S1.servo_start;
S1_MC_MoveVelocity(Execute := _p7, Axis := Sol_kol, Velocity := S1.move_velocity_velocity, Acceleration := S1.move_velocity_acc, Deceleration := S1.move_velocity_dcc, Jerk := S1.move_velocity_jerk, Direction := S1.move_velocity_direction, Continuous := S1.move_velocity_continous, BufferMode := S1.move_velocity_buffermode, Busy => S1.move_velocity_busy, Active => S1.move_velocity_active, CommandAborted => S1.move_velocity_aborted, Error => S1.move_velocity_err, ErrorID => S1.move_velocity_errid);
S1.move_velocity_done := S1_MC_MoveVelocity.InVelocity;
(* Rung 7 *)
_p8 := Sistem_Calisiyor AND S1.pwr_status AND S1.sync_move_start AND S1.servo_start;
S1_MC_SyncMoveAbsolute(Execute := _p8, Axis := Sol_kol, Position := S1.move_position, Direction := S1.move_direction, BufferMode := S1.sync_move_buffer, Busy => S1.sync_move_busy, Active => S1.sync_move_active, CommandAborted => S1.sync_move_aborted, Error => S1.sync_move_error, ErrorID => S1.sync_move_errorid);
S1.sync_move_inPosition := S1_MC_SyncMoveAbsolute.InPosition;
(* Rung 8 *)
_p9 := Sistem_Calisiyor AND S1.pwr_status AND S1.sync_move_relative_start AND S1.servo_start;
S1_MC_SyncMoveVelocity(Execute := _p9, Axis := Sol_kol, Velocity := S1.move_velocity, CmdPosMode := S1_MC_SyncMoveVelocity.CmdPosMode, BufferMode := S1.sync_move_relative_buffer, Busy => S1.sync_move_relative_busy, Active => S1.sync_move_relative_active, CommandAborted => S1.sync_move_relative_aborted, Error => S1.sync_move_relative_error, ErrorID => S1.sync_move_relative_errorid);
S1.sync_move_relative_invelocity := S1_MC_SyncMoveVelocity.InVelocity;
END_PROGRAM